FUNCTION_BLOCK FB_GetObjPropChecksum
VAR_INPUT
	bExecute : BOOL;
END_VAR
VAR_OUTPUT
	bBusy : BOOL;
	nResult : UINT;
END_VAR
VAR
	rTrig			: R_TRIG;
	nCounter		: USINT;
	wPrevChecksum	: WORD;
	nObjChecksum 	: UINT;
	iter			: FB_ObjCollectIteratorDeep;
END_VAR
VAR_IN_OUT
	ObjectDirectoryRef : FB_ObjectDirectory;
END_VAR

rTrig(CLK:= bExecute);
IF rTrig.Q THEN
	bBusy := TRUE;
	wPrevChecksum := 16#FFFF;
	ObjectDirectoryRef.objectList.M_GetIterator(iter);
END_IF

IF bExecute THEN
	nCounter := 0;
	WHILE iter.pNode > 0 AND_THEN iter.pNode^.P_pObject > 0 DO
		nObjChecksum := iter.pNode^.P_pObject^.M_GetPropCheckSum();
		wPrevChecksum := F_DATA_TO_CRC16_CCITT(ADR(nObjChecksum),SIZEOF(nObjChecksum),wPrevChecksum);
		nCounter := nCounter + 1;
		iter.M_Increment();
		IF nCounter = 100 THEN
			RETURN;
		END_IF
	END_WHILE
	nResult := wPrevChecksum;
	bBusy := FALSE;
ELSE
	bBusy := FALSE;
	nResult := 0;
END_IF

END_FUNCTION_BLOCK

(* stored: Version 1.1.0.1, ProductVersion 3.1.4020.12
   POU FB_GetObjPropChecksum: Id {2330becd-0800-4b66-8ac6-23e2154e2b1f}, SpecialFunc None *)
